(* IEC 61131-3 sources: codesys-mcp-toolkit/standalone-sync/sources_st/511_05/PRGs, 7 files *)

(* ---- InfluxUdpSender.prg.st ---- *)
// @OBJECT_ID: 7d4ed387-9382-45d7-b1fe-40ec3c2ade09
// @DECLARATION
PROGRAM InfluxUdpSender
VAR
		fbSender: FB_InfluxUdpSender;
	fbBuf    : FB_InfluxBuffer;
	sendData : STRING(5000); // Data to send
	sIP : STRING :='192.168.150.133'; // InfluxIP
    uiPort : UINT := 8089; // Influx port
	sParam:STRING(200);
END_VAR

// @IMPLEMENTATION
		sendData := 'CEX15,title=aliy2s_app511_abak_101_172 ';

// Initialization (Measurement mariyu Tag set cheyadam)
// =============================================================
fbBuf(sMeasurement:= 'CEX15', sTagKey:= 'title', sTagValue:= 'aliy2s_app511_abak_101_172');

fbBuf.AddReal('rPosValveDiazo',   GVL.gInputRegs.rPosValveDiazo);
fbBuf.AddReal('rPosValveSoda',   GVL.gInputRegs.rPosValveSoda);
fbBuf.AddReal('rPosValveSteam',   GVL.gInputRegs.rPosValveSteam);

fbBuf.AddReal('rPhApp511',   GVL.gInputRegs.rPhApp511);

fbBuf.AddReal('rTempApp511',   GVL.gInputRegs.rTempApp511);

fbBuf.AddReal('WE_1_app_511',   GVL.gInputRegs.WE_1);

fbBuf.AddReal('WE_2_app_511',   GVL.gInputRegs.WE_2);

fbBuf.AddReal('TotalWater_511',   GVL.gInputRegs.IR_TotalWater);

fbBuf.AddReal('TotalSoda_511',   GVL.gInputRegs.IR_TotalSoda);

fbBuf.AddReal('FlowSoda_511',   GVL.gInputRegs.IR_FlowSoda);

fbBuf.AddReal('FlowWater_511',   GVL.gInputRegs.IR_FlowWater);
// Send Data

// =============================================================
fbSender(sSendData:= fbBuf.sBuffer, sIPInflux:= sIP, uiPortInflux:= uiPort);

(* ---- PLC_PRG_MBS_TCP_SLAVE.prg.st ---- *)
// @OBJECT_ID: 87d9b965-00ad-4702-8b83-68f97ffc0669
// @DECLARATION
PROGRAM PLC_PRG_MBS_TCP_SLAVE
VAR
	bFirstLoop	: BOOL := FALSE;
	fbSlv		: AbakPLCUtils.MDB;

	pInputRegs			:	POINTER TO WORD;
	wInputRegsLength	:	WORD 	:= SIZEOF(GVL.gInputRegs)/2;

	pHoldingRegs			:	POINTER TO WORD;
	wHoldingRegsLength	:	WORD 	:= SIZEOF(GVL.gHoldingRegs)/2;

	pInputs			:	POINTER TO BOOL;
	wInputsLength	:	WORD 	:= SIZEOF(GVL.gInputs);

	pCoils			:	POINTER TO BOOL;
	wCoilsLength	:	WORD 	:= SIZEOF(GVL.gCoils);

	wIndex		:	WORD := 0;

	pMbHolding			:	POINTER TO WORD;
	pOldMbHoldingRegs			:	POINTER TO WORD;
	pOldHoldingRegs			:	POINTER TO WORD;

	wMbHolding	:   ARRAY[0..1] OF WORD;
	wOldMbHoldingRegs	:   ARRAY[0..( SIZEOF(GVL.gHoldingRegs)/2-1)] OF WORD;
	wOldHoldingRegs	:   ARRAY[0..(SIZEOF(GVL.gHoldingRegs)/2-1)] OF WORD;

	pMbCoil		:	POINTER TO BOOL;
	pOldMbCoils			:	POINTER TO BOOL;
	pOldCoils			:	POINTER TO BOOL;

	bMbCoil	:   ARRAY[0..0] OF BOOL;
	bOldMbCoils	:   ARRAY[0..(SIZEOF(GVL.gCoils) -1)] OF BOOL;
	bOldCoils	:   ARRAY[0..(SIZEOF(GVL.gCoils) -1)] OF BOOL;

	bIsGetMb: BYTE := 0;

	    wInputRegsOffset    : WORD := 0;  // InputRegs начинаются с адреса 1000
    wInputsOffset       : WORD := 499;   // Inputs начинаются с адреса
    wHoldingRegsOffset  : WORD := 100;     // HoldingRegs - без смещения (или задай своё)
    wCoilsOffset        : WORD := 0;     // Coi
END_VAR

// @IMPLEMENTATION
IF NOT bFirstLoop THEN
	fbSlv.IsVirtualModbus := 0;

	GVL.gInputRegs.INPUTREGS := SIZEOF(GVL.gInputRegs)/2;
	GVL.gInputRegs.HOLDINGS := SIZEOF(GVL.gHoldingRegs)/2;
	GVL.gInputRegs.INPUTS := SIZEOF(GVL.gInputs);
	GVL.gInputRegs.COILS := SIZEOF(GVL.gCoils);

	MBS_HoldingRegs_Change();
	MBS_Coils_Change();

	GVL.gHoldingRegs :=PVL.rHoldingRegs;
	bFirstLoop := TRUE;
ELSE
	MBS_HoldingRegs_Change();
	MBS_Coils_Change();

	MBS_InputRegs_WRITE();
	MBS_Inputs_WRITE();
	PVL.rHoldingRegs :=GVL.gHoldingRegs;
END_IF

(* ---- PRG_Apparatus511.prg.st ---- *)
// @OBJECT_ID: 9f480724-c0be-439f-90b3-2c3ccbb6fbf9
// @DECLARATION
PROGRAM PRG_Apparatus511
VAR
    // Экземпляр функционального блока управления клапаном пара
    fbSteamControl_511 : FB_UniversalSteamValveControl;

    // Переменные для связи с HMI (если они еще не заданы в GVL)
    xEnableTempControl : BOOL;  // Команда с HMI: Включить автоматическое поддержание температуры
    rTempSetpoint_511  : REAL;  // Задание поддерживаемой температуры в аппарате (до 100 °C)
    xResetTempPID      : BOOL;  // Команда сброса ошибки ПИД-регулятора

    // Промежуточная переменная для связи флагов режима
    xSteamAutoMode     : BOOL;  // TRUE = АВТО, FALSE = РУЧНОЙ
END_VAR

// @IMPLEMENTATION
// --- ВЫЗОВ БЛОКА ПОДДЕРЖАНИЯ ТЕМПЕРАТУРЫ АППАРАТА 511 ---

fbSteamControl_511(
    xEnable       := xEnableTempControl,          // Команда оператора на запуск контура
    rTempActual   := GVL.gInputRegs.rTempApp511,  // Текущая температура из аппарата 511 [3, 4]
    rSetpoint     := rTempSetpoint_511,           // Уставка температуры (до 100 °C) [5, 6]
    xReset        := xResetTempPID,               // Сброс ПИД
    rKp           := GVL.gHoldingRegs.rKp_Steam_511,
    rTn           := GVL.gHoldingRegs.rTn_Steam_511,
    rTv           := GVL.gHoldingRegs.rTv_Steam_511,
    rLimitLow     := 0.0,
    rLimitHigh    := 100.0,

    // IN_OUT переменные (передаются по ссылке напрямую)
    rValveOut     := GVL.gHoldingRegs.rAutoSet_Steam, // Запись выхода ПИД в авто-задание клапана пара [1, 2]
    xAutoModeCmd  := xSteamAutoMode                   // Получаем команду режима от ФБ
);

// --- СИНХРОНИЗАЦИЯ РЕЖИМОВ УПРАВЛЕНИЯ ---
// Согласно вашей логике, клапан пара (fbValveSteam) работает в ручном режиме
// когда GVL.gCoils.xManualMode_Steam = TRUE [2].
// Поскольку наш ФБ выдает TRUE для режима АВТО, нам нужно инвертировать этот сигнал:
GVL.gCoils.xManualMode_Steam := NOT xSteamAutoMode;

(* ---- PRG_Apparatus511_CascadeDrain.prg.st ---- *)
// @OBJECT_ID: c5ea459a-3d8c-4dff-9b4c-b4e64976f6c9
// @DECLARATION
PROGRAM PRG_Apparatus511_CascadeDrain
VAR
    // Экземпляр последней версии блока (с конечным автоматом)
    fbCascadeDrain511 : FB_AutoCouplingDrainCascade;

    // Вспомогательные переменные для инверсии ручного/автоматического режимов
    xDiazoAutoMode    : BOOL;
    xSodaAutoMode     : BOOL;
END_VAR

// @IMPLEMENTATION

// --- 1. ВЫЗОВ АЛГОРИТМА СЛИВА С ПОДДЕРЖАНИЕМ pH ---
fbCascadeDrain511(
    // Управление
    xStart             := GVL.gCoils.xStartCoupling_511,

    // Параметры Диазосоединения
    rFlowDiazoActual   := GVL.gInputRegs.IR_FlowDiazo,         // Мгновенный расход [1]
    rFlowDiazoSetpoint := GVL.gHoldingRegs.rSetFlowDiazo_511,  // Уставка расхода [1]

    // Параметры pH
    rPhActual          := GVL.gInputRegs.rPhApp511,            // Показания pH-метра [1]
    rPhSetpoint        := GVL.gHoldingRegs.rSetPh_511,         // Целевая уставка pH [1]

    // Настройки условия завершения (конвертация UINT секунд в TIME)
    rZeroFlowThreshold := GVL.gHoldingRegs.rZeroFlowThreshold_511,
    tEmptyDelay        := UDINT_TO_TIME(UINT_TO_UDINT(GVL.gHoldingRegs.uiEmptyDelaySec_511) * 1000),

    // Настройки ПИД
    rKp_Diazo          := GVL.gHoldingRegs.rKp_Diazo_511,
    rTn_Diazo          := GVL.gHoldingRegs.rTn_Diazo_511,
    rKp_pH             := GVL.gHoldingRegs.rKp_pH_511,
    rTn_pH             := GVL.gHoldingRegs.rTn_pH_511,

    // Прямая связь с авто-заданиями физических клапанов (IN_OUT)
    rValveOutDiazo     := GVL.gHoldingRegs.rAutoSet_Diazo,     // [3]
    xAutoModeCmdDiazo  := xDiazoAutoMode,

    rValveOutSoda      := GVL.gHoldingRegs.rAutoSet_Soda,      // [3]
    xAutoModeCmdSoda   := xSodaAutoMode
);

// --- 2. СИНХРОНИЗАЦИЯ РЕЖИМОВ (Ручной/Авто) ---
// В физической логике клапанов TRUE = Ручной режим, поэтому инвертируем команду от блока
GVL.gCoils.xManualMode_Diazo := NOT xDiazoAutoMode;
GVL.gCoils.xManualMode_Soda  := NOT xSodaAutoMode;

// --- 3. ПЕРЕДАЧА СТАТУСОВ КОНЕЧНОГО АВТОМАТА НА HMI ---
// Булевые лампочки состояния процесса
GVL.gCoils.xCouplingActive_511 := fbCascadeDrain511.xActive;
GVL.gCoils.xCouplingDone_511   := fbCascadeDrain511.xDone;

// Числовые коды, оставшееся время и текст
GVL.gInputRegs.rTimeLeft_511   := fbCascadeDrain511.rTimeLeft;  // Оставшиеся секунды при падении расхода
GVL.gInputRegs.rStateCode_511  := fbCascadeDrain511.rStateCode; // 0.0, 1.0, 2.0, 3.0, 4.0
GVL.sStateStr_511              := fbCascadeDrain511.sStateStr;  // Расшифровка этапа

(* ---- PRG_Apparatus511_Heating.prg.st ---- *)
// @OBJECT_ID: 7ad46e98-502c-4d9e-a2ee-bf251bb90bbe
// @DECLARATION
PROGRAM PRG_Apparatus511_Heating
VAR
    // Экземпляр нашего блока автоматического нагрева
    fbAutoHeater511 : FB_AutoHeater;

    // Вспомогательная переменная для связи флагов режима клапана
    xSteamAutoMode  : BOOL;
END_VAR

// @IMPLEMENTATION
// --- Автоматический нагрев аппарата 511 ---
fbAutoHeater511(
// --- Входы управления с HMI ---
xStart        := GVL.gCoils.xStartHeating_511,      // Признак запуска нагрева с панели оператора
xKeepTemp     := GVL.gCoils.xKeepTempHeating_511,   // TRUE = поддерживать температуру после достижения
rTargetTemp   := GVL.gHoldingRegs.rSetTempApp511,   // Уставка целевой температуры (до 100 °C)
// --- Технологические параметры ---
rTempActual   := GVL.gInputRegs.rTempApp511,        // Фактическая температура в емкости
rTolerance    := 0.5,                               // Допуск в градусах
// --- Настройки пид ---
rKp           := GVL.gHoldingRegs.rKp_Steam_511,
rTn           := GVL.gHoldingRegs.rTn_Steam_511,
rTv           := GVL.gHoldingRegs.rTv_Steam_511,
// --- Выходы на исполнительные механизмы (IN_OUT) ---
rValveOut     := GVL.gHoldingRegs.rAutoSet_Steam,
xAutoModeCmd  := xSteamAutoMode
);

(* ---- PRG_ModbusSlave_Sync.prg.st ---- *)
// @OBJECT_ID: 808e203d-1a0e-46f1-b7a1-0b905523bfa3
// @DECLARATION
(*
* @fb: PRG_ModbusSlave_Sync
* @desc: Исправленная синхронизация через прямые указатели (устранение C0047/C0077)
*)
PROGRAM PRG_ModbusSlave_Sync
VAR
    fbSlv               : abakplcutils.MDB;
    sStatus             : STRING(255);

    // Вспомогательные буферы
    wMbHolding          : ARRAY[0..500] OF WORD;
    wOldMbHolding       : ARRAY[0..500] OF WORD;

    // Указатели для работы со структурами GVL как с массивами
    pCurrWord           : POINTER TO WORD;
    pOldWord            : POINTER TO WORD;

    wIndex              : WORD;
    uiHoldRegsCnt       : WORD;
    uiInRegsCnt         : WORD;
    xFirstLoop          : BOOL := TRUE;

    C_INPUT_REG_START   : WORD := 1;
    C_HOLD_REG_START    : WORD := 1000;
END_VAR

// @IMPLEMENTATION
// 1. Инициализация и расчет длин (через SIZEOF, чтобы не зависеть от типов)
IF xFirstLoop THEN
    uiInRegsCnt   := ANY_TO_WORD(SIZEOF(GVL.gInputRegs) / 2);
    uiHoldRegsCnt := ANY_TO_WORD(SIZEOF(GVL.gHoldingRegs) / 2);

    // Предзаполнение Modbus и локального зеркала (используем SysMem для скорости)
    fbSlv.SetWordRegs(reg := C_HOLD_REG_START, pBuf := ADR(GVL.gHoldingRegs), cnt := uiHoldRegsCnt);
    SysMem.SysMemCpy(pDest := ADR(wOldMbHolding), pSrc := ADR(GVL.gHoldingRegs), udiCount := uiHoldRegsCnt * 2);

    xFirstLoop := FALSE;
    RETURN;
END_IF

// --- ШАГ 1: Input Registers (Запись всей структуры целиком через указатель) ---
sStatus := 'Обновление Input Registers';
fbSlv.SetWordRegs(reg := C_INPUT_REG_START, pBuf := ADR(GVL.gInputRegs), cnt := uiInRegsCnt);

// --- ШАГ 2: Holding Registers (Синхронизация через пошаговый доступ к памяти) ---
sStatus := 'Синхронизация Holding...';
fbSlv.GetWordRegs(reg := C_HOLD_REG_START, pBuf := ADR(wMbHolding), cnt := uiHoldRegsCnt);

FOR wIndex := 0 TO (uiHoldRegsCnt - 1) DO
    // Получаем адреса текущего слова в GVL и в нашем зеркале Old
    pCurrWord := ADR(GVL.gHoldingRegs) + (wIndex * 2); // Смещение в байтах (WORD = 2 байта)
    pOldWord  := ADR(wOldMbHolding) + (wIndex * 2);

    // Сценарий А: Изменение в ПЛК
    IF pCurrWord^ <> pOldWord^ THEN
        fbSlv.SetWord(reg := C_HOLD_REG_START + wIndex, val := pCurrWord^);
        pOldWord^ := pCurrWord^; // Обновляем зеркало

    // Сценарий Б: Изменение в Modbus (от SCADA)
    ELSIF wMbHolding[wIndex] <> pOldWord^ THEN
        pCurrWord^ := wMbHolding[wIndex]; // Пишем напрямую в структуру GVL
        pOldWord^  := wMbHolding[wIndex]; // Обновляем зеркало
    END_IF
END_FOR

// Синхронизация с энергонезависимой памятью
PVL.rHoldingRegs := GVL.gHoldingRegs;

(* ---- PRG_Valves.prg.st ---- *)
// @OBJECT_ID: 4a778488-a136-43da-a5b5-63d2fca365f4
// @DECLARATION
PROGRAM PRG_Valves
VAR

    // Экземпляры логики управления для каждого клапана
    fbValveDiazo : FB_ValveLogic;
    fbValveSoda  : FB_ValveLogic;
    fbValveSteam : FB_ValveLogic;

    // Флаг для однократной инициализации указателей
    xInitDone    : BOOL := FALSE;
    // Экземпляр функционального блока для клапана подачи воды
    fbWaterValve : FB_ValveS_Compact;

END_VAR

// @IMPLEMENTATION
// --- 1. ОДНОКРАТНАЯ ИНИЦИАЛИЗАЦИЯ (Привязка адресов) ---
IF NOT xInitDone THEN

    // Привязка для клапана Диазосоединения
    fbValveDiazo.Init(
        pManualVar := ADR(gvl.gHoldingRegs.rValveManSet_Diazo),       // Уставка с HMI
        pAutoVar   := ADR(gvl.gHoldingRegs.rAutoSet_Diazo),     // Уставка от ПИД/Логики
        pOutputVar := ADR(gvl.gHoldingRegs.AO1_CmdValveDiazo)       // Физический выход (M2)
    );

    // Привязка для клапана Едкого натра (Соды)
    fbValveSoda.Init(
        pManualVar := ADR(gvl.gHoldingRegs.rValveManSet_Soda),
        pAutoVar   := ADR(gvl.gHoldingRegs.rAutoSet_Soda),
        pOutputVar := ADR(gvl.gHoldingRegs.AO2_CmdValveSoda)        // Физический выход (M2)
    );

    // Привязка для клапана Пара
    fbValveSteam.Init(
        pManualVar := ADR(gvl.gHoldingRegs.rValveManSet_Steam),
        pAutoVar   := ADR(gvl.gHoldingRegs.rAutoSet_Steam),
        pOutputVar := ADR(gvl.gHoldingRegs.AO3_CmdValveSteam)       // Физический выход (M2)
    );

    xInitDone := TRUE;
END_IF;

// --- 2. ЦИКЛИЧЕСКИЙ ВЫЗОВ ЛОГИКИ ---

// Управление клапаном Диазосоединения
fbValveDiazo(
    xModeManual :=gvl.gCoils.xManualMode_Diazo,
    rMinLimit   := 0.0,
    rMaxLimit   := 100.0
);

// Управление клапаном Едкого натра
fbValveSoda(
    xModeManual := gvl.gCoils.xManualMode_Soda,
    rMinLimit   := 0.0,
    rMaxLimit   := 100.0
);

// Управление клапаном Пара
fbValveSteam(
    xModeManual := gvl.gCoils.xManualMode_Steam,
    rMinLimit   := 0.0,
    rMaxLimit   := 100.0
);

// Вызов блока управления водяным клапаном
fbWaterValve(
    xMode        := gvl.gCoils.xWaterValve_AutoMode,
    xManControl  := gvl.gcoils.xWaterValve_HmiOpen,
    xAutoControl := gvl.gcoils.xWaterValve_AutoReq,
    xOutControl  => gvl.gInputs.xWaterValve_Out
);
